{attribute 'qualified_only' := ''}
{attribute 'strict' := ''}
{attribute 'to_string' := ''}
TYPE cLaneSel :
(
	None := 0,
	Green := 1,
	Red := 2,
	Blue := 3
);
END_TYPE

(* stored: Version 1.1.0.1, ProductVersion 3.1.4024.6
   DUT cLaneSel: Id {e9195ac5-0a1b-4b64-b3d6-5b469630e14e} *)
